Fanuc KAREL source: kt00098.KL

PROGRAM KT00098
%STACKSIZE=65535
%PRIORITY=65535
%NOLOCKGROUP
VAR
I1 : INTEGER
I2 : INTEGER
OUT : REAL
BEGIN
I1=2
I2=3
I1=2
I2=3
-- UNSAFE_SOURCE_IR line 12: OUT = (int_to_real(I1) / int_to_real(I2))
END KT00098
